FUNCTION alg_g_z: LREAL
{ S7_Optimized_Access := 'true' }
    VAR_INPUT
        state: STATE;
    END_VAR

BEGIN
    alg_g_z := state.curTime;
END_FUNCTION
